// TwinCAT 3 PLC project PlcMSC500
// ProgramVersion: 3.1.4024.0
// libraries:
//   Tc2_Standard, * (Beckhoff Automation GmbH)
//   Tc2_System, * (Beckhoff Automation GmbH)
//   Tc2_TcpIp, * (Beckhoff Automation GmbH)
//   Tc3_Module, * (Beckhoff Automation GmbH)
// project tree:
//   / PlcTask.TcTTO
//   POUs/ FB_MSC_Client.TcPOU, MAIN.TcPOU
// real-time tasks:
//   TASK PlcMSC: cycle T#10ms, priority 20, ADS port 350
//   TASK PlcAsyril: cycle T#10ms, priority 21, ADS port 351

CONFIGURATION PlcMSC500
    RESOURCE PLC ON TwinCAT3
        TASK PlcTask(INTERVAL := T#10ms, PRIORITY := 20);
        PROGRAM MAIN WITH PlcTask : MAIN;
    END_RESOURCE
END_CONFIGURATION

// ---- POUs/MAIN.TcPOU
PROGRAM MAIN
VAR
	bInit: BOOL := TRUE;
	fbSocketCloseAll: FB_SocketCloseAll; 
	bSocketCloseError: BOOL;
	nSocketCloseError: UDINT;
	
		fbFBMSCFB_MSC_Client		: FB_MSC_Client;
		sClient1SendData			: STRING(255) := 'ActivateRobot';					// Auszuführender Befehl
		nServer1Port				: UDINT 				:= 10000;					// Port des Geräts
		sServer1Host				: T_IPv4Addr 			:= '192.168.1.20'; 			// IP des Geräts
		bStartClient1Communication	: BOOL 					:= TRUE;
		tClient1CycleTime			: TIME 					:= T#0.5S;
		bClient1SendTrigger			: BOOL;
		bClient1Connected			: BOOL;
		sClient1ReceivedData		: STRING(255);										// Antwort
		bClient1Busy				: BOOL;
		bClientError1				: BOOL;
		nClient1ErrorID1			: UDINT;		
		bReady						: BOOL;												// Trigger

END_VAR

IF bInit THEN 				// Init Step to close all sockets after login PLC with  downlaod
	fbSocketCloseAll(
		sSrvNetId:= '', 
		bExecute:= TRUE, 
		tTimeout:= T#3S, 
		bBusy=> , 
		bError=> bSocketCloseError, 
		nErrId=> nSocketCloseError);
	IF NOT (fbSocketCloseAll.bBusy OR fbSocketCloseAll.bError) THEN
		bInit := FALSE;
		fbSocketCloseAll(bExecute:= FALSE);
	END_IF
ELSE
	
	fbFBMSCFB_MSC_Client(
		nRemotePort:= nServer1Port, 								// Server port
		sRemoteHost:= sServer1Host, 								// Server IP (empty for local communication)
		bStartCommunication:= bStartClient1Communication, 			// Start communication, when FALSE, connection is closed
		sSendData:= sClient1SendData, 								// Data that are sent to the server
		tCycleTimeSend:= (*tClient1CycleTime*), 					// TimeInterval for cyclic sending
		bSendTrigger:= ,											// Trigger to send one telegramm manually 
		bConnected => bClient1Connected,							// Switches to TRUE when Client is connected to a server
		sReceivedData=> sClient1ReceivedData,						// Data that are received
		bBusy=> bClient1Busy, 
		bError=> bClientError1, 
		nErrorID=> nClient1ErrorID1, ); 
	
	IF bClient1Connected THEN
		IF bReady  THEN
			sClient1SendData;
			fbFBMSCFB_MSC_Client.bSendTrigger := TRUE;
		ELSE
			fbFBMSCFB_MSC_Client.bSendTrigger := FALSE;
		END_IF
		bReady := FALSE;
	END_IF 
		

END_IF

END_PROGRAM

// ---- POUs/FB_MSC_Client.TcPOU
FUNCTION_BLOCK FB_MSC_Client
VAR_INPUT
	sRemoteHost: T_IPv4Addr;
	nRemotePort: UDINT;
	sSendData: STRING(255);	
	bStartCommunication: BOOL;
	tCycleTimeSend: TIME;
	bSendTrigger : BOOL;
END_VAR
VAR_OUTPUT
	bConnected: BOOL;
	sReceivedData: STRING(255);
	nErrorID: UDINT;
	bError: BOOL;
	bBusy: BOOL;
END_VAR
VAR
	iState: INT;
	fbSocketConnect: FB_SocketConnect;
	fbSocketSend: FB_SocketSend;
	fbSocketClose: FB_SocketClose;
	fbSocketReceive: FB_SocketReceive;
	hSocket: T_HSOCKET;

	fbTimer: TON;
	nRecBytes: UDINT;
	bExecuteSocketSend: BOOL;
	RTrig: R_TRIG;
END_VAR

CASE iState OF
0:	// Init State
	fbSocketConnect(bExecute := FALSE); 
	fbSocketSend(bExecute := FALSE); 
	fbSocketReceive(bExecute := FALSE);
	fbSocketClose(bExecute := FALSE); 
	bConnected := FALSE; 
	bBusy := FALSE;
	IF bStartCommunication = TRUE THEN									// Start communication manually 
		iState := iState + 10;
		bBusy := TRUE;
		bError := FALSE;
	END_IF

10:	// Connect Server
	fbSocketConnect(													// Open connection to server
		sSrvNetId:= '', 
		sRemoteHost:= sRemoteHost, 
		nRemotePort:= nRemotePort, 
		bExecute:= TRUE, 
		tTimeout:= T#4S, 
		bBusy=> , 
		bError=> bError, 
		nErrId=> nErrorID, 
		hSocket=> hSocket);

	IF hSocket.handle <> 0 AND NOT (fbSocketConnect.bBusy) THEN			// Handle is created
		bConnected := TRUE; 
		iState :=iState + 5;
	ELSIF bError THEN
		iState := 0; 	
	END_IF
	
	
15:																		// StartCommunication
	IF (tCycleTimeSend <> T#0MS) THEN									// Send data cyclically
		fbTimer(IN:= NOT fbTimer.Q, PT:= tCycleTimeSend, Q=> , ET=> );		
	END_IF
	RTrig(CLK:= bSendTrigger, Q=> );									// SendData on manuel trigger
	
	fbSocketSend(														// Send Data
		sSrvNetId:= '', 
		hSocket:= hSocket, 
		cbLen:= SIZEOF(sSendData), 
		pSrc:= ADR(sSendData), 
		bExecute:= (fbTimer.Q OR RTrig.Q), 
		tTimeout:= T#2S, 
		bError=> bError, 
		nErrId=> nErrorID, 
		nErrId=> );

	fbSocketReceive(													// ReceiveData
		sSrvNetId:= '', 
		hSocket:= hSocket, 
		cbLen:= SIZEOF(sReceivedData), 
		pDest:=  ADR(sReceivedData), 
		bExecute:= true, 
		tTimeout:= T#3S, 
		bBusy=> , 
		bError=> bError, 
		nErrId=> nErrorID, 
		nRecBytes=> nRecBytes);
		
	IF NOT fbSocketReceive.bBusy THEN									// Check cyclically for new data
		fbSocketReceive(bExecute := FALSE);
	END_IF						
	IF NOT bStartCommunication OR bError THEN							// Close connection in case of error or manual communication stop
		iState := 20;
	END_IF
20: 
	fbSocketClose(														// Close connection
		sSrvNetId:= '', 
		hSocket:= hSocket, 
		bExecute:= TRUE, 
		tTimeout:= T#4S, 
		bBusy=> , 
		bError=> bError, 
		nErrId=> nErrorID );
	IF NOT fbSocketClose.bBusy THEN
		iState :=0;		
	END_IF
END_CASE

END_FUNCTION_BLOCK
